FUNCTION proj48_TupleStruct_5: LREAL
VAR_INPUT
    tuple: TupleStruct_5;
END_VAR


        proj48_TupleStruct_5 := tuple.field48;

END_FUNCTION

(* stored: ProductVersion 3.1.0.18, Version 1.1.0.1 *)
